{attribute 'GeneratedUsingTerminal: EK1122-0000-0018'}
{attribute addProperty BoxType "EK1122-0000-0018"}
{attribute addProperty Id "Beckhoff_EP9xxxsub_EK1100EK1100_1FC0878B2A_0001_EP9128_0020_0016A_0001_EP9128_0020_0016_F00690F4593"}
{attribute addProperty CRC "783209979"}
{attribute addProperty Size "595"}
TYPE Beckhoff_EP9xxxEK1122_2EAED5FB EXTENDS EK1122_1FC0878B :
STRUCT
	{attribute addProperty Name "Beckhoff_EP9xxxsub_EK1100"}
	{attribute addProperty PreviousPort "Beckhoff EP9xxxEK1122 : D"}
	Beckhoff_EP9xxxsub_EK1100 : EK1100_1FC0878B;
	{attribute addProperty Name "A_0001_EP9128_0020_0016"}
	{attribute addProperty PreviousPort "Beckhoff EP9xxxsub EK1100 : C"}
	A_0001_EP9128_0020_0016 : A_0001_EP9128_0020_0016_F00690F4;
END_STRUCT
END_TYPE

(* stored: Version 1.2.0.0, ProductVersion 3.1.4024.9
   DUT Beckhoff_EP9xxxEK1122_2EAED5FB: Id {5631ac24-c95e-4ade-8e27-a45398e7d6bc} *)
